(*
A circular queue implementation for managing `I_Arg`.  
*)
INTERFACE I_ArgQueue EXTENDS I_Debug

(*
Returns the current head index of the queue, indicating the next position for insertion.
*)
PROPERTY Head : UDINT
GET
END_GET
END_PROPERTY

(*
Provides access to the underlying list structure that holds the queue's argument objects.
*)
PROPERTY List : I_ArgList
GET
END_GET
END_PROPERTY

(*
Returns the current tail index of the queue, indicating the next position for retrieval.
*)
PROPERTY Tail : UDINT
GET
END_GET
END_PROPERTY

END_INTERFACE

(* stored: Version 1.1.0.1
   Itf I_ArgQueue: Id {479af9a2-73ee-4633-80f3-a7501838f2f1}
   Property Head: Id {63cffb29-df17-41ec-a017-453383157af9}
   Get Get: Id {7b0919ac-80d0-4104-a8ee-5c8b397efa95}
   Property List: Id {22d13380-699e-45b5-956e-33b334fa798a}
   Get Get: Id {8bd18bf7-b6ad-434a-927e-8b900b9a1b7d}
   Property Tail: Id {044d209c-e47e-44ea-85f2-0bbbbbf8c740}
   Get Get: Id {b2840707-759f-40f0-b9d2-b3d1e79747d1} *)
